{attribute 'qualified_only'}
{attribute 'strict'}
TYPE E_RS_COMMAND :
(
	NONE	:= 0,
	
	RESET,
	INIT,
	STOP,
	ENABLE,
	DISABLE,
	
	READ,
	READ_USER,
	MONITOR,
	MONITOR_USER,
	STOPMON,
	
	CTRL_CMD
	
);
END_TYPE

(* stored: Version 1.1.0.1, ProductVersion 3.1.4024.3
   DUT E_RS_COMMAND: Id {9f1b0375-7f99-4abd-93ac-793147a81243} *)
